// TIA Portal V19 export
FUNCTION "FC_FW_Auftrag_Step2_KB" : Void   // FC1082, LAD
TITLE = Schritt CM03/CM04 -> CM01/CM02
{ S7_Optimized_Access := 'TRUE' }
// Ältesten Warenträger in CM03/CM04 suchen und nach CM01/CM02 transportieren
// stored: AutoNumber false, SetENOAutomatically false
   VAR_INPUT
      Frg_Schritt : Bool;
   END_VAR
   VAR_OUTPUT
      nextStep : Bool;
      startStep : Bool;
      parkStep : Bool;
   END_VAR
   VAR_IN_OUT
      Quelle : Int;
      Ziel : Int;
      Positionen : Array[1..30] of "UDT_Auftrag_Pos";
   END_VAR
   VAR_TEMP
      Sperre_Kurz_li_CM01 : Bool;
      Sperre_Kurz_re_CM01 : Bool;
      Sperre_Lang_CM01 : Bool;
      Sperre_Kurz_li_CM02 : Bool;
      Sperre_Kurz_re_CM02 : Bool;
      Sperre_Lang_CM02 : Bool;
      Vorzug : Bool;
      Vorzug1 : Bool;
      Vorzug2 : Bool;
      Befehl_ok : Bool;
      tmpQuelle : Int;
      Oldest : Real;
   END_VAR
   VAR CONSTANT
      Wt_Cmd_AetzenCM01 : Int := 1;
      Wt_Cmd_AetzenCM02 : Int := 13;
   END_VAR
BEGIN

REGION Network 1 (SCL)
   IF (#Quelle <> 0) AND (#Ziel <> 0) THEN
       #nextStep := #Positionen[#Quelle].Sperre;
       #startStep := NOT #nextStep;
       #Quelle := 0;
       #Ziel := 0;
       RETURN;
   END_IF;

   #Quelle := 0;
   #Ziel := 0;
   #nextStep := FALSE;
   #startStep := FALSE;

   IF NOT #Frg_Schritt THEN
       #nextStep := TRUE;
       RETURN;
   END_IF;
END_REGION

REGION Network 2 (SCL): Positionen sperren
   // GO nur "161"
   //Groß links nicht möglich
   #Positionen[9].CheckSperre := (#Positionen[3].Sperre ) OR (#Positionen[9].Wt_Cmd <> #Wt_Cmd_AetzenCM01);

   //Groß rechts nicht möglich
   #Positionen[10].CheckSperre := (#Positionen[4].Sperre AND #Positionen[16].Sperre) OR (#Positionen[10].Wt_Cmd <> #Wt_Cmd_AetzenCM01);

   //kein Platz für Kurz links in CM01
   #Sperre_Kurz_li_CM01 := #Positionen[1].Sperre AND #Positionen[5].Sperre;

   //kein Platz für Kurz links in CM02
   #Sperre_Kurz_li_CM02 := #Positionen[13].Sperre AND #Positionen[17].Sperre;

   //kein Platz für Kurz rechts in CM01
   #Sperre_Kurz_re_CM01 := #Positionen[2].Sperre AND #Positionen[6].Sperre;

   //kein Platz für Kurz rechts in CM02
   #Sperre_Kurz_re_CM02 := #Positionen[14].Sperre AND #Positionen[18].Sperre;

   //kein Platz für Lang in CM01
   #Sperre_Lang_CM01 := (#Positionen[1].Sperre OR #Positionen[2].Sperre) AND (#Positionen[5].Sperre OR #Positionen[6].Sperre);

   //kein Platz für Lang in CM02
   #Sperre_Lang_CM02:= (#Positionen[13].Sperre OR #Positionen[14].Sperre) AND (#Positionen[17].Sperre OR #Positionen[18].Sperre);

   //Lang in P7 oder
   //kein Platz auf rechter Seite
   //-> P8 sperren
   #Positionen[8].CheckSperre := #Sperre_Kurz_re_CM01 OR (#Positionen[7].Wt_Typ = "WT_Typ_LS") OR (#Positionen[8].Wt_Cmd <> #Wt_Cmd_AetzenCM01);

   //Lang in P7 und kein Platz für Lang oder
   //kein Platz auf linker Seite
   //-> P7 sperren
   #Positionen[7].CheckSperre := #Sperre_Kurz_li_CM01 OR ((#Positionen[7].Wt_Typ = "WT_Typ_LS") AND #Sperre_Lang_CM01) OR (#Positionen[7].Wt_Cmd <> #Wt_Cmd_AetzenCM01);

   //Lang in P7 oder
   //kein Platz auf rechter Seite
   //-> P12 sperren
   #Positionen[12].CheckSperre := #Sperre_Kurz_re_CM01 OR (#Positionen[11].Wt_Typ = "WT_Typ_LS") OR (#Positionen[12].Wt_Cmd <> #Wt_Cmd_AetzenCM01);

   //Lang in P11 und kein Platz für Lang oder
   //kein Platz auf linker Seite
   //-> P11 sperren
   #Positionen[11].CheckSperre := #Sperre_Kurz_li_CM01 OR ((#Positionen[11].Wt_Typ = "WT_Typ_LS") AND #Sperre_Lang_CM01) OR (#Positionen[11].Wt_Cmd <> #Wt_Cmd_AetzenCM01);

   //Lang in P19 oder
   //kein Platz auf rechter Seite
   //-> P20 sperren
   #Positionen[20].CheckSperre := #Sperre_Kurz_re_CM02 OR (#Positionen[19].Wt_Typ = "WT_Typ_LS") OR (#Positionen[20].Wt_Cmd <> #Wt_Cmd_AetzenCM02);

   //Lang in P19 und kein Platz für Lang oder
   //kein Platz auf linker Seite
   //-> P19 sperren
   #Positionen[19].CheckSperre := #Sperre_Kurz_li_CM02 OR ((#Positionen[19].Wt_Typ = "WT_Typ_LS") AND #Sperre_Lang_CM02) OR (#Positionen[19].Wt_Cmd <> #Wt_Cmd_AetzenCM02);

   //Lang in P23 oder
   //kein Platz auf rechter Seite
   //-> P24 sperren
   #Positionen[24].CheckSperre := #Sperre_Kurz_re_CM02 OR (#Positionen[23].Wt_Typ = "WT_Typ_LS") OR (#Positionen[24].Wt_Cmd <> #Wt_Cmd_AetzenCM02);

   //Lang in P23 und kein Platz für Lang oder
   //kein Platz auf linker Seite
   //-> P23 sperren
   #Positionen[23].CheckSperre := #Sperre_Kurz_li_CM02 OR ((#Positionen[23].Wt_Typ = "WT_Typ_LS") AND #Sperre_Lang_CM02) OR (#Positionen[23].Wt_Cmd <> #Wt_Cmd_AetzenCM02);
END_REGION

REGION Network 3 (SCL): Ältesten WT suchen
   //
   #Oldest := 0;
   #tmpQuelle := 0;

   //CM03
   "FC_FW_Auftrag_Suche"(Pos1 := 7,
                         Pos2 := 12,
                         Positionen := #Positionen,
                         Quelle := #tmpQuelle,
                         Oldest := #Oldest);

   //CM04
   "FC_FW_Auftrag_Suche"(Pos1 := 19,
                         Pos2 := 24,
                         Positionen := #Positionen,
                         Quelle := #tmpQuelle,
                         Oldest := #Oldest);
END_REGION

REGION Network 4 (SCL): Auswertung
   IF #tmpQuelle = 0 THEN
       //kein WT
       #nextStep := TRUE;
       RETURN;
   END_IF;

   IF NOT #Positionen[#tmpQuelle].Fertig THEN
       #parkStep := TRUE;
       RETURN;
   END_IF;

   IF (#tmpQuelle = 9) THEN
       //Gross links nur "161"
       IF NOT #Positionen[3].Sperre THEN
           "FC_FW_Auftrag_Befehl"(inQuelle := #tmpQuelle,
                                  inZiel := 3,
                                  Befehl_ok => #Befehl_ok,
                                  outQuelle => #Quelle,
                                  outZiel => #Ziel);

           #nextStep := NOT #Befehl_ok;
       ELSE
           #nextStep := TRUE;
       END_IF;
       RETURN;
   END_IF;

   IF (#tmpQuelle = 10) THEN
       //Gross rechts nur "161"
       IF NOT #Positionen[4].Sperre THEN
           "FC_FW_Auftrag_Befehl"(inQuelle := #tmpQuelle,
                                  inZiel := 4,
                                  Befehl_ok => #Befehl_ok,
                                  outQuelle => #Quelle,
                                  outZiel => #Ziel);

           #nextStep := NOT #Befehl_ok;
       ELSE
           #nextStep := TRUE;
       END_IF;
       RETURN;
   END_IF;

   IF (#Positionen[#tmpQuelle].Wt_Typ = "WT_Typ_LS") AND ((#tmpQuelle = 7) OR (#tmpQuelle = 11)) THEN
       //Lang "161"
       IF NOT #Positionen[5].Sperre AND NOT #Positionen[6].Sperre THEN
           "FC_FW_Auftrag_Befehl"(inQuelle := #tmpQuelle,
                                  inZiel := 5,
                                  Befehl_ok => #Befehl_ok,
                                  outQuelle => #Quelle,
                                  outZiel => #Ziel);

           #nextStep := NOT #Befehl_ok;
       ELSIF NOT #Positionen[1].Sperre AND NOT #Positionen[2].Sperre THEN
           "FC_FW_Auftrag_Befehl"(inQuelle := #tmpQuelle,
                                  inZiel := 1,
                                  Befehl_ok => #Befehl_ok,
                                  outQuelle => #Quelle,
                                  outZiel => #Ziel);

           #nextStep := NOT #Befehl_ok;
       ELSE
           #nextStep := TRUE;
       END_IF;
       RETURN;
   END_IF;

   IF (#Positionen[#tmpQuelle].Wt_Typ = "WT_Typ_LS") AND ((#tmpQuelle = 19) OR (#tmpQuelle = 23)) THEN
       //Lang "151"
       IF NOT #Positionen[17].Sperre AND NOT #Positionen[18].Sperre THEN
           "FC_FW_Auftrag_Befehl"(inQuelle := #tmpQuelle,
                                  inZiel := 17,
                                  Befehl_ok => #Befehl_ok,
                                  outQuelle => #Quelle,
                                  outZiel => #Ziel);

           #nextStep := NOT #Befehl_ok;
       ELSIF NOT #Positionen[13].Sperre AND NOT #Positionen[14].Sperre THEN
           "FC_FW_Auftrag_Befehl"(inQuelle := #tmpQuelle,
                                  inZiel := 13,
                                  Befehl_ok => #Befehl_ok,
                                  outQuelle => #Quelle,
                                  outZiel => #Ziel);

           #nextStep := NOT #Befehl_ok;
       ELSE
           #nextStep := TRUE;
       END_IF;
       RETURN;
   END_IF;

   IF (#tmpQuelle = 7) OR (#tmpQuelle = 11) THEN
       //Kurz links "161"
       #Vorzug1 := NOT #Positionen[1].Sperre AND #Positionen[2].Sperre;
       #Vorzug2 := NOT #Positionen[5].Sperre AND #Positionen[6].Sperre;

       #Vorzug := NOT #Vorzug2 AND #Vorzug1;
       IF NOT #Positionen[5].Sperre AND NOT #Vorzug THEN
           "FC_FW_Auftrag_Befehl"(inQuelle := #tmpQuelle,
                                  inZiel := 5,
                                  Befehl_ok => #Befehl_ok,
                                  outQuelle => #Quelle,
                                  outZiel => #Ziel);

           #nextStep := NOT #Befehl_ok;
           RETURN;
       END_IF;

       #Vorzug := NOT #Vorzug1 AND #Vorzug1;
       IF NOT #Positionen[1].Sperre AND NOT #Vorzug THEN
           "FC_FW_Auftrag_Befehl"(inQuelle := #tmpQuelle,
                                  inZiel := 1,
                                  Befehl_ok => #Befehl_ok,
                                  outQuelle => #Quelle,
                                  outZiel => #Ziel);

           #nextStep := NOT #Befehl_ok;
           RETURN;
       END_IF;

       #nextStep := TRUE;
       RETURN;
   END_IF;

   IF (#tmpQuelle = 8) OR (#tmpQuelle = 12) THEN
       //Kurz rechts "161"
       #Vorzug1 := NOT #Positionen[2].Sperre AND #Positionen[1].Sperre;
       #Vorzug2 := NOT #Positionen[6].Sperre AND #Positionen[5].Sperre;

       #Vorzug := NOT #Vorzug2 AND #Vorzug1;
       IF NOT #Positionen[6].Sperre AND NOT #Vorzug THEN
           "FC_FW_Auftrag_Befehl"(inQuelle := #tmpQuelle,
                                  inZiel := 6,
                                  Befehl_ok => #Befehl_ok,
                                  outQuelle => #Quelle,
                                  outZiel => #Ziel);

           #nextStep := NOT #Befehl_ok;
           RETURN;
       END_IF;


       #Vorzug := NOT #Vorzug1 AND #Vorzug2;
       IF NOT #Positionen[2].Sperre AND NOT #Vorzug THEN
           "FC_FW_Auftrag_Befehl"(inQuelle := #tmpQuelle,
                                  inZiel := 2,
                                  Befehl_ok => #Befehl_ok,
                                  outQuelle => #Quelle,
                                  outZiel => #Ziel);

           #nextStep := NOT #Befehl_ok;
           RETURN;
       END_IF;

       #nextStep := TRUE;
       RETURN;
   END_IF;

   IF (#tmpQuelle = 19) OR (#tmpQuelle = 23) THEN
       //Kurz links "151"
       #Vorzug1 := NOT #Positionen[13].Sperre AND #Positionen[14].Sperre;
       #Vorzug2 := NOT #Positionen[17].Sperre AND #Positionen[18].Sperre;

       #Vorzug := NOT #Vorzug2 AND #Vorzug1;
       IF NOT #Positionen[17].Sperre AND NOT #Vorzug THEN
           "FC_FW_Auftrag_Befehl"(inQuelle := #tmpQuelle,
                                  inZiel := 17,
                                  Befehl_ok => #Befehl_ok,
                                  outQuelle => #Quelle,
                                  outZiel => #Ziel);

           #nextStep := NOT #Befehl_ok;
           RETURN;
       END_IF;

       #Vorzug := NOT #Vorzug1 AND #Vorzug1;
       IF NOT #Positionen[13].Sperre AND NOT #Vorzug THEN
           "FC_FW_Auftrag_Befehl"(inQuelle := #tmpQuelle,
                                  inZiel := 13,
                                  Befehl_ok => #Befehl_ok,
                                  outQuelle => #Quelle,
                                  outZiel => #Ziel);

           #nextStep := NOT #Befehl_ok;
           RETURN;
       END_IF;

       #nextStep := TRUE;
       RETURN;
   END_IF;

   IF (#tmpQuelle = 20) OR (#tmpQuelle = 24) THEN
       //Kurz rechts "151"
       #Vorzug1 := NOT #Positionen[2].Sperre AND #Positionen[1].Sperre;
       #Vorzug2 := NOT #Positionen[6].Sperre AND #Positionen[5].Sperre;

       #Vorzug := NOT #Vorzug2 AND #Vorzug1;
       IF NOT #Positionen[18].Sperre AND NOT #Vorzug THEN
           "FC_FW_Auftrag_Befehl"(inQuelle := #tmpQuelle,
                                  inZiel := 18,
                                  Befehl_ok => #Befehl_ok,
                                  outQuelle => #Quelle,
                                  outZiel => #Ziel);

           #nextStep := NOT #Befehl_ok;
           RETURN;
       END_IF;

       #Vorzug := NOT #Vorzug1 AND #Vorzug2;
       IF NOT #Positionen[14].Sperre AND NOT #Vorzug THEN
           "FC_FW_Auftrag_Befehl"(inQuelle := #tmpQuelle,
                                  inZiel := 14,
                                  Befehl_ok => #Befehl_ok,
                                  outQuelle => #Quelle,
                                  outZiel => #Ziel);

           #nextStep := NOT #Befehl_ok;
           RETURN;
       END_IF;

       #nextStep := TRUE;
       RETURN;
   END_IF;

   //
   #nextStep := TRUE;
END_REGION
END_FUNCTION
